FUNCTION makeTupleStruct_3: TupleStruct_3
VAR_INPUT
    field0: BOOL;
    field1: BOOL;
    field2: BOOL;
    field3: BOOL;
    field4: BOOL;
    field5: BOOL;
    field6: BOOL;
    field7: BOOL;
    field8: BOOL;
    field9: BOOL;
    field10: BOOL;
    field11: BOOL;
    field12: BOOL;
    field13: BOOL;
    field14: BOOL;
    field15: BOOL;
    field16: BOOL;
    field17: BOOL;
    field18: BOOL;
    field19: BOOL;
    field20: BOOL;
    field21: BOOL;
    field22: BOOL;
    field23: BOOL;
    field24: BOOL;
    field25: BOOL;
    field26: BOOL;
    field27: BOOL;
    field28: BOOL;
    field29: BOOL;
    field30: BOOL;
    field31: BOOL;
    field32: BOOL;
    field33: BOOL;
    field34: BOOL;
    field35: BOOL;
    field36: BOOL;
    field37: BOOL;
    field38: BOOL;
    field39: BOOL;
    field40: BOOL;
    field41: BOOL;
    field42: BOOL;
    field43: BOOL;
    field44: BOOL;
    field45: BOOL;
    field46: BOOL;
    field47: BOOL;
    field48: BOOL;
    field49: BOOL;
    field50: BOOL;
    field51: BOOL;
    field52: BOOL;
    field53: BOOL;
    field54: BOOL;
    field55: BOOL;
    field56: BOOL;
    field57: BOOL;
    field58: BOOL;
    field59: BOOL;
    field60: BOOL;
    field61: BOOL;
    field62: BOOL;
    field63: BOOL;
    field64: BOOL;
    field65: BOOL;
    field66: BOOL;
    field67: BOOL;
    field68: BOOL;
    field69: BOOL;
    field70: BOOL;
    field71: BOOL;
    field72: BOOL;
    field73: BOOL;
    field74: BOOL;
    field75: BOOL;
    field76: BOOL;
    field77: BOOL;
    field78: BOOL;
    field79: BOOL;
    field80: BOOL;
    field81: BOOL;
    field82: BOOL;
    field83: BOOL;
    field84: BOOL;
    field85: BOOL;
    field86: BOOL;
    field87: BOOL;
    field88: BOOL;
    field89: BOOL;
    field90: BOOL;
    field91: BOOL;
    field92: BOOL;
    field93: BOOL;
    field94: BOOL;
    field95: BOOL;
    field96: BOOL;
    field97: BOOL;
    field98: BOOL;
    field99: BOOL;
END_VAR
VAR
    rslt: TupleStruct_3;
END_VAR


        rslt.field0 := field0;
rslt.field1 := field1;
rslt.field2 := field2;
rslt.field3 := field3;
rslt.field4 := field4;
rslt.field5 := field5;
rslt.field6 := field6;
rslt.field7 := field7;
rslt.field8 := field8;
rslt.field9 := field9;
rslt.field10 := field10;
rslt.field11 := field11;
rslt.field12 := field12;
rslt.field13 := field13;
rslt.field14 := field14;
rslt.field15 := field15;
rslt.field16 := field16;
rslt.field17 := field17;
rslt.field18 := field18;
rslt.field19 := field19;
rslt.field20 := field20;
rslt.field21 := field21;
rslt.field22 := field22;
rslt.field23 := field23;
rslt.field24 := field24;
rslt.field25 := field25;
rslt.field26 := field26;
rslt.field27 := field27;
rslt.field28 := field28;
rslt.field29 := field29;
rslt.field30 := field30;
rslt.field31 := field31;
rslt.field32 := field32;
rslt.field33 := field33;
rslt.field34 := field34;
rslt.field35 := field35;
rslt.field36 := field36;
rslt.field37 := field37;
rslt.field38 := field38;
rslt.field39 := field39;
rslt.field40 := field40;
rslt.field41 := field41;
rslt.field42 := field42;
rslt.field43 := field43;
rslt.field44 := field44;
rslt.field45 := field45;
rslt.field46 := field46;
rslt.field47 := field47;
rslt.field48 := field48;
rslt.field49 := field49;
rslt.field50 := field50;
rslt.field51 := field51;
rslt.field52 := field52;
rslt.field53 := field53;
rslt.field54 := field54;
rslt.field55 := field55;
rslt.field56 := field56;
rslt.field57 := field57;
rslt.field58 := field58;
rslt.field59 := field59;
rslt.field60 := field60;
rslt.field61 := field61;
rslt.field62 := field62;
rslt.field63 := field63;
rslt.field64 := field64;
rslt.field65 := field65;
rslt.field66 := field66;
rslt.field67 := field67;
rslt.field68 := field68;
rslt.field69 := field69;
rslt.field70 := field70;
rslt.field71 := field71;
rslt.field72 := field72;
rslt.field73 := field73;
rslt.field74 := field74;
rslt.field75 := field75;
rslt.field76 := field76;
rslt.field77 := field77;
rslt.field78 := field78;
rslt.field79 := field79;
rslt.field80 := field80;
rslt.field81 := field81;
rslt.field82 := field82;
rslt.field83 := field83;
rslt.field84 := field84;
rslt.field85 := field85;
rslt.field86 := field86;
rslt.field87 := field87;
rslt.field88 := field88;
rslt.field89 := field89;
rslt.field90 := field90;
rslt.field91 := field91;
rslt.field92 := field92;
rslt.field93 := field93;
rslt.field94 := field94;
rslt.field95 := field95;
rslt.field96 := field96;
rslt.field97 := field97;
rslt.field98 := field98;
rslt.field99 := field99;
makeTupleStruct_3 := rslt;

END_FUNCTION

(* stored: ProductVersion 3.1.0.18, Version 1.1.0.1 *)
